PROGRAM Touchpanel
VAR
	bContactAvailable AT %I*: BOOL;
	rXadc AT %I*: REAL;
	rYadc AT %I*: REAL;
	rZadc AT %I*: REAL;
	iXadc AT %I*: INT;
	iYadc AT %I*: INT;
	iZadc AT %I*: INT;
	rMaxTouchPosX: REAL := 363 / 2;
	rMaxTouchPosY: REAL := 294 / 2;
	touch_scale_x: TOUCH_SCALE;
	touch_scale_y: TOUCH_SCALE;
	
END_VAR

VAR CONSTANT
	iStep AT %Q*: INT := 1010;
	rQ_Kalman AT %Q*: REAL := 1.0;  
	rR_Kalman AT %Q*: REAL := 400.0;
END_VAR

touch_scale_x(rX:=rXadc, 
              rDistance:=363.0, 
              rMinAdc:=100, 
              rMaxAdc:=3890,
			  rOffset:=rMaxTouchPosX);
				 
touch_scale_y(rX:=rYadc, 
              rDistance:=286.0, 
              rMinAdc:=100, 
              rMaxAdc:=3900,
			  rOffset:=rMaxTouchPosY);

END_PROGRAM

(* stored: Version 1.1.0.1, ProductVersion 3.1.4024.12
   POU Touchpanel: Id {8959fee0-1d1f-4cda-8331-278bca6d8d02}, SpecialFunc None *)
